REGION Network 47: ACTION IN LOADING CELL UNIT 2
   RUNG wire#powerrail
      "FC17900_MAINTENANCE_SEQUENCE"(REQUEST := 0, NUMBER_STEPS := 3, FIRST_STEP_DONE := "DB17000_MAINTENANCE_GLOBAL_VARIABLES".ACTION_DONE.POWDER.UNIT_2.HOPPER_1.LOAD_CELLS, SECOND_STEP_DONE := "DB17000_MAINTENANCE_GLOBAL_VARIABLES".ACTION_DONE.POWDER.UNIT_2.HOPPER_2.LOAD_CELLS, THRID_STEP_DONE := "DB17000_MAINTENANCE_GLOBAL_VARIABLES".ACTION_DONE.POWDER.UNIT_2.HOPPER_3.LOAD_CELLS, FOURTH_STEP_DONE := 0, FIFTH_STEP_DONE := 0, SIXTH_STEP_DONE := 0, SEVENTH_STEP_DONE := 0, FIRST_OPERATOR_HELP => "DB17100_MAINTENANCE_OPERATOR_HELP".OPERATOR_HELP[36], SECOND_OPERATOR_HELP => "DB17100_MAINTENANCE_OPERATOR_HELP".OPERATOR_HELP[41], THRID_OPERATOR_HELP => "DB17100_MAINTENANCE_OPERATOR_HELP".OPERATOR_HELP[46], FOURTH_OPERATOR_HELP => #NULL, FIFTH_OPERATOR_HELP => #NULL, SIXTH_OPERATOR_HELP => #NULL, SEVENTH_OPERATOR_HELP => #NULL, MAINTENANCE_IN_PROGRESS => "DB17200_MAINTENANCE_SEQUENCE".MAINTENANCE_IN_PROGRESS[42])
   END_RUNG
   // the same network as SCL:
   "FC17900_MAINTENANCE_SEQUENCE"(REQUEST := 0,
                           NUMBER_STEPS := 3,
                           FIRST_STEP_DONE := "DB17000_MAINTENANCE_GLOBAL_VARIABLES".ACTION_DONE.POWDER.UNIT_2.HOPPER_1.LOAD_CELLS,
                           SECOND_STEP_DONE := "DB17000_MAINTENANCE_GLOBAL_VARIABLES".ACTION_DONE.POWDER.UNIT_2.HOPPER_2.LOAD_CELLS,
                           THRID_STEP_DONE := "DB17000_MAINTENANCE_GLOBAL_VARIABLES".ACTION_DONE.POWDER.UNIT_2.HOPPER_3.LOAD_CELLS,
                           FOURTH_STEP_DONE := 0,
                           FIFTH_STEP_DONE := 0,
                           SIXTH_STEP_DONE := 0,
                           SEVENTH_STEP_DONE := 0,
                           FIRST_OPERATOR_HELP => "DB17100_MAINTENANCE_OPERATOR_HELP".OPERATOR_HELP[36],
                           SECOND_OPERATOR_HELP => "DB17100_MAINTENANCE_OPERATOR_HELP".OPERATOR_HELP[41],
                           THRID_OPERATOR_HELP => "DB17100_MAINTENANCE_OPERATOR_HELP".OPERATOR_HELP[46],
                           FOURTH_OPERATOR_HELP => #NULL,
                           FIFTH_OPERATOR_HELP => #NULL,
                           SIXTH_OPERATOR_HELP => #NULL,
                           SEVENTH_OPERATOR_HELP => #NULL,
                           MAINTENANCE_IN_PROGRESS => "DB17200_MAINTENANCE_SEQUENCE".MAINTENANCE_IN_PROGRESS[42]);
END_REGION

REGION Network 48: COMPLETE CHANGE OF FEEDER UNIT 1
   RUNG wire#powerrail
      "FC17900_MAINTENANCE_SEQUENCE"(REQUEST := 0, NUMBER_STEPS := 3, FIRST_STEP_DONE := "DB17000_MAINTENANCE_GLOBAL_VARIABLES".ACTION_DONE.POWDER.UNIT_1.FEEDER_1.TIGHTNESS_TEST_L1, SECOND_STEP_DONE := "DB17000_MAINTENANCE_GLOBAL_VARIABLES".ACTION_DONE.POWDER.UNIT_1.FEEDER_1.TIGHTNESS_TEST_L2, THRID_STEP_DONE := "DB17000_MAINTENANCE_GLOBAL_VARIABLES".ACTION_DONE.POWDER.UNIT_1.GENERAL.POWDER_FLOW_OBTAINING, FOURTH_STEP_DONE := 0, FIFTH_STEP_DONE := 0, SIXTH_STEP_DONE := 0, SEVENTH_STEP_DONE := 0, FIRST_OPERATOR_HELP => "DB17100_MAINTENANCE_OPERATOR_HELP".OPERATOR_HELP[22], SECOND_OPERATOR_HELP => "DB17100_MAINTENANCE_OPERATOR_HELP".OPERATOR_HELP[23], THRID_OPERATOR_HELP => "DB17100_MAINTENANCE_OPERATOR_HELP".OPERATOR_HELP[6], FOURTH_OPERATOR_HELP => #NULL, FIFTH_OPERATOR_HELP => #NULL, SIXTH_OPERATOR_HELP => #NULL, SEVENTH_OPERATOR_HELP => #NULL, MAINTENANCE_IN_PROGRESS => "DB17200_MAINTENANCE_SEQUENCE".MAINTENANCE_IN_PROGRESS[43])
   END_RUNG
   // the same network as SCL:
   "FC17900_MAINTENANCE_SEQUENCE"(REQUEST := 0,
                           NUMBER_STEPS := 3,
                           FIRST_STEP_DONE := "DB17000_MAINTENANCE_GLOBAL_VARIABLES".ACTION_DONE.POWDER.UNIT_1.FEEDER_1.TIGHTNESS_TEST_L1,
                           SECOND_STEP_DONE := "DB17000_MAINTENANCE_GLOBAL_VARIABLES".ACTION_DONE.POWDER.UNIT_1.FEEDER_1.TIGHTNESS_TEST_L2,
                           THRID_STEP_DONE := "DB17000_MAINTENANCE_GLOBAL_VARIABLES".ACTION_DONE.POWDER.UNIT_1.GENERAL.POWDER_FLOW_OBTAINING,
                           FOURTH_STEP_DONE := 0,
                           FIFTH_STEP_DONE := 0,
                           SIXTH_STEP_DONE := 0,
                           SEVENTH_STEP_DONE := 0,
                           FIRST_OPERATOR_HELP => "DB17100_MAINTENANCE_OPERATOR_HELP".OPERATOR_HELP[22],
                           SECOND_OPERATOR_HELP => "DB17100_MAINTENANCE_OPERATOR_HELP".OPERATOR_HELP[23],
                           THRID_OPERATOR_HELP => "DB17100_MAINTENANCE_OPERATOR_HELP".OPERATOR_HELP[6],
                           FOURTH_OPERATOR_HELP => #NULL,
                           FIFTH_OPERATOR_HELP => #NULL,
                           SIXTH_OPERATOR_HELP => #NULL,
                           SEVENTH_OPERATOR_HELP => #NULL,
                           MAINTENANCE_IN_PROGRESS => "DB17200_MAINTENANCE_SEQUENCE".MAINTENANCE_IN_PROGRESS[43]);
END_REGION

REGION Network 49: COMPLETE CHANGE OF FEEDER UNIT 2
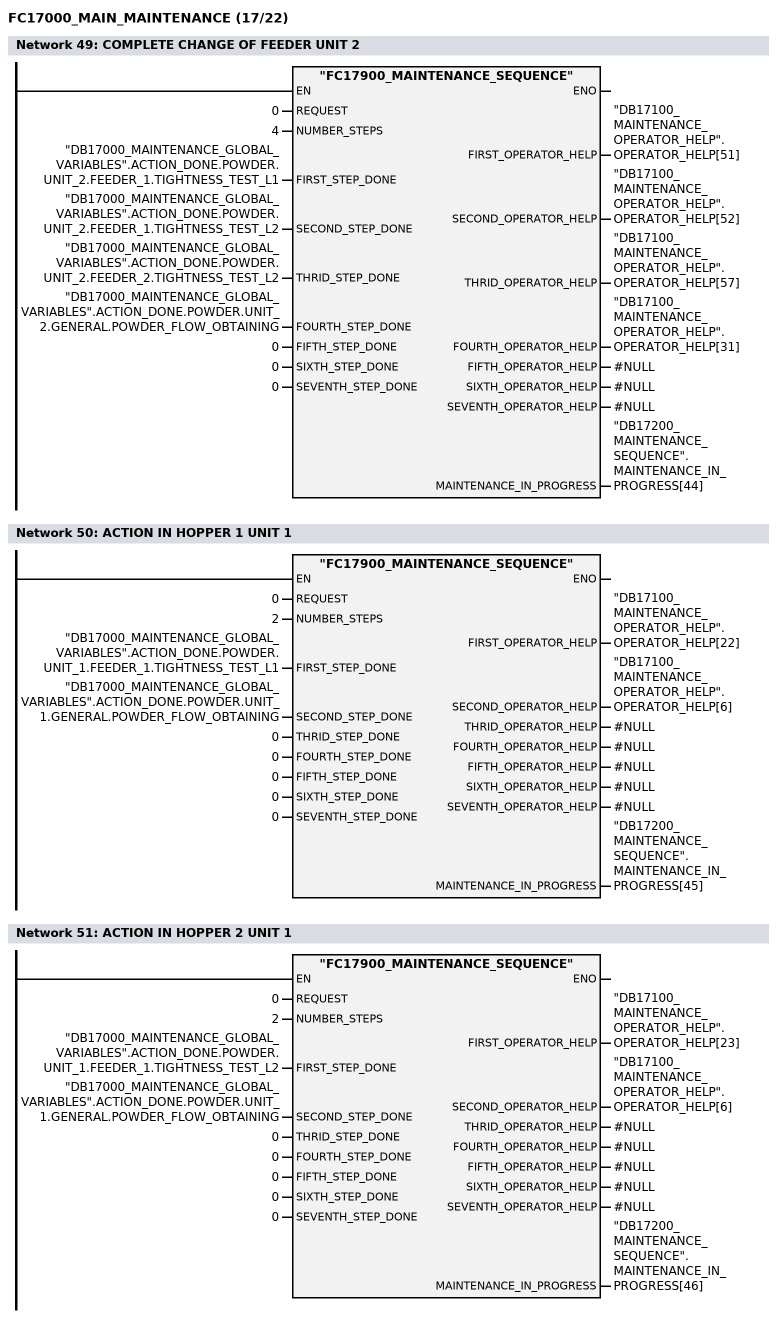
   RUNG wire#powerrail
      "FC17900_MAINTENANCE_SEQUENCE"(REQUEST := 0, NUMBER_STEPS := 4, FIRST_STEP_DONE := "DB17000_MAINTENANCE_GLOBAL_VARIABLES".ACTION_DONE.POWDER.UNIT_2.FEEDER_1.TIGHTNESS_TEST_L1, SECOND_STEP_DONE := "DB17000_MAINTENANCE_GLOBAL_VARIABLES".ACTION_DONE.POWDER.UNIT_2.FEEDER_1.TIGHTNESS_TEST_L2, THRID_STEP_DONE := "DB17000_MAINTENANCE_GLOBAL_VARIABLES".ACTION_DONE.POWDER.UNIT_2.FEEDER_2.TIGHTNESS_TEST_L2, FOURTH_STEP_DONE := "DB17000_MAINTENANCE_GLOBAL_VARIABLES".ACTION_DONE.POWDER.UNIT_2.GENERAL.POWDER_FLOW_OBTAINING, FIFTH_STEP_DONE := 0, SIXTH_STEP_DONE := 0, SEVENTH_STEP_DONE := 0, FIRST_OPERATOR_HELP => "DB17100_MAINTENANCE_OPERATOR_HELP".OPERATOR_HELP[51], SECOND_OPERATOR_HELP => "DB17100_MAINTENANCE_OPERATOR_HELP".OPERATOR_HELP[52], THRID_OPERATOR_HELP => "DB17100_MAINTENANCE_OPERATOR_HELP".OPERATOR_HELP[57], FOURTH_OPERATOR_HELP => "DB17100_MAINTENANCE_OPERATOR_HELP".OPERATOR_HELP[31], FIFTH_OPERATOR_HELP => #NULL, SIXTH_OPERATOR_HELP => #NULL, SEVENTH_OPERATOR_HELP => #NULL, MAINTENANCE_IN_PROGRESS => "DB17200_MAINTENANCE_SEQUENCE".MAINTENANCE_IN_PROGRESS[44])
   END_RUNG
   // the same network as SCL:
   "FC17900_MAINTENANCE_SEQUENCE"(REQUEST := 0,
                           NUMBER_STEPS := 4,
                           FIRST_STEP_DONE := "DB17000_MAINTENANCE_GLOBAL_VARIABLES".ACTION_DONE.POWDER.UNIT_2.FEEDER_1.TIGHTNESS_TEST_L1,
                           SECOND_STEP_DONE := "DB17000_MAINTENANCE_GLOBAL_VARIABLES".ACTION_DONE.POWDER.UNIT_2.FEEDER_1.TIGHTNESS_TEST_L2,
                           THRID_STEP_DONE := "DB17000_MAINTENANCE_GLOBAL_VARIABLES".ACTION_DONE.POWDER.UNIT_2.FEEDER_2.TIGHTNESS_TEST_L2,
                           FOURTH_STEP_DONE := "DB17000_MAINTENANCE_GLOBAL_VARIABLES".ACTION_DONE.POWDER.UNIT_2.GENERAL.POWDER_FLOW_OBTAINING,
                           FIFTH_STEP_DONE := 0,
                           SIXTH_STEP_DONE := 0,
                           SEVENTH_STEP_DONE := 0,
                           FIRST_OPERATOR_HELP => "DB17100_MAINTENANCE_OPERATOR_HELP".OPERATOR_HELP[51],
                           SECOND_OPERATOR_HELP => "DB17100_MAINTENANCE_OPERATOR_HELP".OPERATOR_HELP[52],
                           THRID_OPERATOR_HELP => "DB17100_MAINTENANCE_OPERATOR_HELP".OPERATOR_HELP[57],
                           FOURTH_OPERATOR_HELP => "DB17100_MAINTENANCE_OPERATOR_HELP".OPERATOR_HELP[31],
                           FIFTH_OPERATOR_HELP => #NULL,
                           SIXTH_OPERATOR_HELP => #NULL,
                           SEVENTH_OPERATOR_HELP => #NULL,
                           MAINTENANCE_IN_PROGRESS => "DB17200_MAINTENANCE_SEQUENCE".MAINTENANCE_IN_PROGRESS[44]);
END_REGION

REGION Network 50: ACTION IN HOPPER 1 UNIT 1
   RUNG wire#powerrail
      "FC17900_MAINTENANCE_SEQUENCE"(REQUEST := 0, NUMBER_STEPS := 2, FIRST_STEP_DONE := "DB17000_MAINTENANCE_GLOBAL_VARIABLES".ACTION_DONE.POWDER.UNIT_1.FEEDER_1.TIGHTNESS_TEST_L1, SECOND_STEP_DONE := "DB17000_MAINTENANCE_GLOBAL_VARIABLES".ACTION_DONE.POWDER.UNIT_1.GENERAL.POWDER_FLOW_OBTAINING, THRID_STEP_DONE := 0, FOURTH_STEP_DONE := 0, FIFTH_STEP_DONE := 0, SIXTH_STEP_DONE := 0, SEVENTH_STEP_DONE := 0, FIRST_OPERATOR_HELP => "DB17100_MAINTENANCE_OPERATOR_HELP".OPERATOR_HELP[22], SECOND_OPERATOR_HELP => "DB17100_MAINTENANCE_OPERATOR_HELP".OPERATOR_HELP[6], THRID_OPERATOR_HELP => #NULL, FOURTH_OPERATOR_HELP => #NULL, FIFTH_OPERATOR_HELP => #NULL, SIXTH_OPERATOR_HELP => #NULL, SEVENTH_OPERATOR_HELP => #NULL, MAINTENANCE_IN_PROGRESS => "DB17200_MAINTENANCE_SEQUENCE".MAINTENANCE_IN_PROGRESS[45])
   END_RUNG
   // the same network as SCL:
   "FC17900_MAINTENANCE_SEQUENCE"(REQUEST := 0,
                           NUMBER_STEPS := 2,
                           FIRST_STEP_DONE := "DB17000_MAINTENANCE_GLOBAL_VARIABLES".ACTION_DONE.POWDER.UNIT_1.FEEDER_1.TIGHTNESS_TEST_L1,
                           SECOND_STEP_DONE := "DB17000_MAINTENANCE_GLOBAL_VARIABLES".ACTION_DONE.POWDER.UNIT_1.GENERAL.POWDER_FLOW_OBTAINING,
                           THRID_STEP_DONE := 0,
                           FOURTH_STEP_DONE := 0,
                           FIFTH_STEP_DONE := 0,
                           SIXTH_STEP_DONE := 0,
                           SEVENTH_STEP_DONE := 0,
                           FIRST_OPERATOR_HELP => "DB17100_MAINTENANCE_OPERATOR_HELP".OPERATOR_HELP[22],
                           SECOND_OPERATOR_HELP => "DB17100_MAINTENANCE_OPERATOR_HELP".OPERATOR_HELP[6],
                           THRID_OPERATOR_HELP => #NULL,
                           FOURTH_OPERATOR_HELP => #NULL,
                           FIFTH_OPERATOR_HELP => #NULL,
                           SIXTH_OPERATOR_HELP => #NULL,
                           SEVENTH_OPERATOR_HELP => #NULL,
                           MAINTENANCE_IN_PROGRESS => "DB17200_MAINTENANCE_SEQUENCE".MAINTENANCE_IN_PROGRESS[45]);
END_REGION

REGION Network 51: ACTION IN HOPPER 2 UNIT 1
   RUNG wire#powerrail
      "FC17900_MAINTENANCE_SEQUENCE"(REQUEST := 0, NUMBER_STEPS := 2, FIRST_STEP_DONE := "DB17000_MAINTENANCE_GLOBAL_VARIABLES".ACTION_DONE.POWDER.UNIT_1.FEEDER_1.TIGHTNESS_TEST_L2, SECOND_STEP_DONE := "DB17000_MAINTENANCE_GLOBAL_VARIABLES".ACTION_DONE.POWDER.UNIT_1.GENERAL.POWDER_FLOW_OBTAINING, THRID_STEP_DONE := 0, FOURTH_STEP_DONE := 0, FIFTH_STEP_DONE := 0, SIXTH_STEP_DONE := 0, SEVENTH_STEP_DONE := 0, FIRST_OPERATOR_HELP => "DB17100_MAINTENANCE_OPERATOR_HELP".OPERATOR_HELP[23], SECOND_OPERATOR_HELP => "DB17100_MAINTENANCE_OPERATOR_HELP".OPERATOR_HELP[6], THRID_OPERATOR_HELP => #NULL, FOURTH_OPERATOR_HELP => #NULL, FIFTH_OPERATOR_HELP => #NULL, SIXTH_OPERATOR_HELP => #NULL, SEVENTH_OPERATOR_HELP => #NULL, MAINTENANCE_IN_PROGRESS => "DB17200_MAINTENANCE_SEQUENCE".MAINTENANCE_IN_PROGRESS[46])
   END_RUNG
   // the same network as SCL:
   "FC17900_MAINTENANCE_SEQUENCE"(REQUEST := 0,
                           NUMBER_STEPS := 2,
                           FIRST_STEP_DONE := "DB17000_MAINTENANCE_GLOBAL_VARIABLES".ACTION_DONE.POWDER.UNIT_1.FEEDER_1.TIGHTNESS_TEST_L2,
                           SECOND_STEP_DONE := "DB17000_MAINTENANCE_GLOBAL_VARIABLES".ACTION_DONE.POWDER.UNIT_1.GENERAL.POWDER_FLOW_OBTAINING,
                           THRID_STEP_DONE := 0,
                           FOURTH_STEP_DONE := 0,
                           FIFTH_STEP_DONE := 0,
                           SIXTH_STEP_DONE := 0,
                           SEVENTH_STEP_DONE := 0,
                           FIRST_OPERATOR_HELP => "DB17100_MAINTENANCE_OPERATOR_HELP".OPERATOR_HELP[23],
                           SECOND_OPERATOR_HELP => "DB17100_MAINTENANCE_OPERATOR_HELP".OPERATOR_HELP[6],
                           THRID_OPERATOR_HELP => #NULL,
                           FOURTH_OPERATOR_HELP => #NULL,
                           FIFTH_OPERATOR_HELP => #NULL,
                           SIXTH_OPERATOR_HELP => #NULL,
                           SEVENTH_OPERATOR_HELP => #NULL,
                           MAINTENANCE_IN_PROGRESS => "DB17200_MAINTENANCE_SEQUENCE".MAINTENANCE_IN_PROGRESS[46]);
END_REGION

REGION Network 52: ACTION IN HOPPER 1 UNIT 2
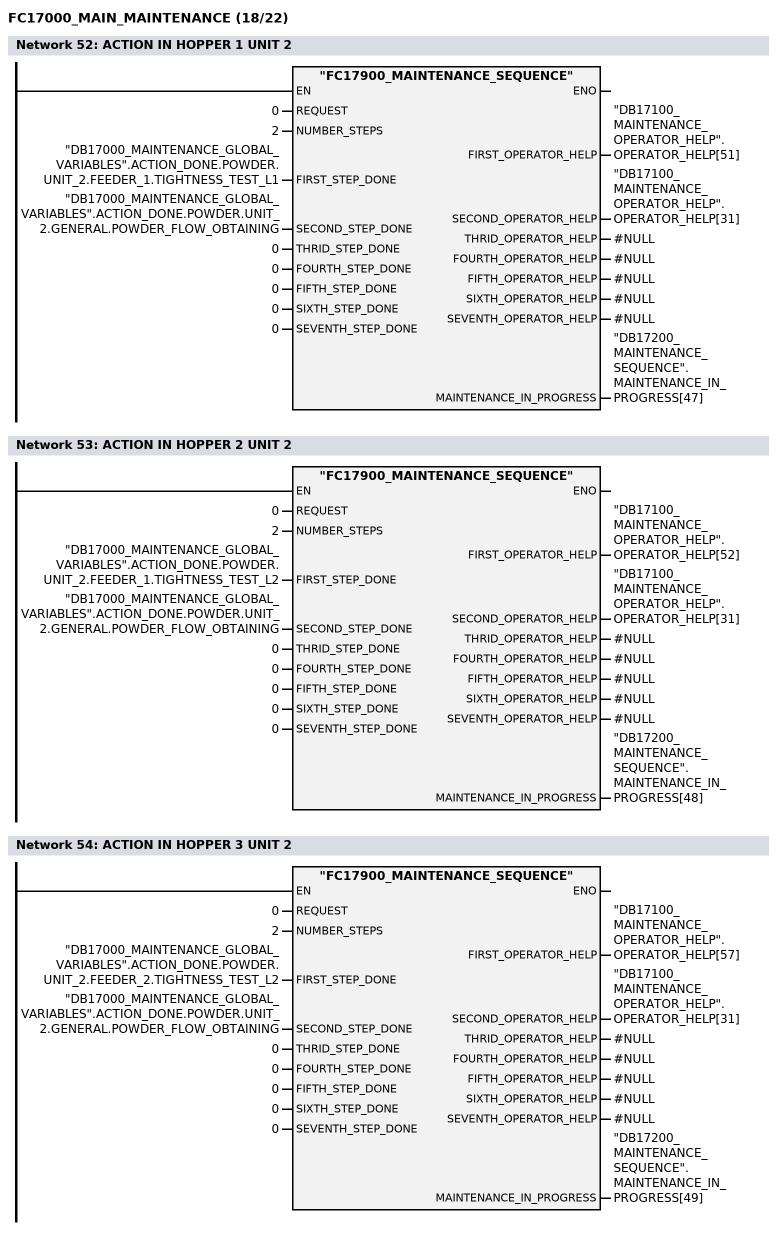
   RUNG wire#powerrail
      "FC17900_MAINTENANCE_SEQUENCE"(REQUEST := 0, NUMBER_STEPS := 2, FIRST_STEP_DONE := "DB17000_MAINTENANCE_GLOBAL_VARIABLES".ACTION_DONE.POWDER.UNIT_2.FEEDER_1.TIGHTNESS_TEST_L1, SECOND_STEP_DONE := "DB17000_MAINTENANCE_GLOBAL_VARIABLES".ACTION_DONE.POWDER.UNIT_2.GENERAL.POWDER_FLOW_OBTAINING, THRID_STEP_DONE := 0, FOURTH_STEP_DONE := 0, FIFTH_STEP_DONE := 0, SIXTH_STEP_DONE := 0, SEVENTH_STEP_DONE := 0, FIRST_OPERATOR_HELP => "DB17100_MAINTENANCE_OPERATOR_HELP".OPERATOR_HELP[51], SECOND_OPERATOR_HELP => "DB17100_MAINTENANCE_OPERATOR_HELP".OPERATOR_HELP[31], THRID_OPERATOR_HELP => #NULL, FOURTH_OPERATOR_HELP => #NULL, FIFTH_OPERATOR_HELP => #NULL, SIXTH_OPERATOR_HELP => #NULL, SEVENTH_OPERATOR_HELP => #NULL, MAINTENANCE_IN_PROGRESS => "DB17200_MAINTENANCE_SEQUENCE".MAINTENANCE_IN_PROGRESS[47])
   END_RUNG
   // the same network as SCL:
   "FC17900_MAINTENANCE_SEQUENCE"(REQUEST := 0,
                           NUMBER_STEPS := 2,
                           FIRST_STEP_DONE := "DB17000_MAINTENANCE_GLOBAL_VARIABLES".ACTION_DONE.POWDER.UNIT_2.FEEDER_1.TIGHTNESS_TEST_L1,
                           SECOND_STEP_DONE := "DB17000_MAINTENANCE_GLOBAL_VARIABLES".ACTION_DONE.POWDER.UNIT_2.GENERAL.POWDER_FLOW_OBTAINING,
                           THRID_STEP_DONE := 0,
                           FOURTH_STEP_DONE := 0,
                           FIFTH_STEP_DONE := 0,
                           SIXTH_STEP_DONE := 0,
                           SEVENTH_STEP_DONE := 0,
                           FIRST_OPERATOR_HELP => "DB17100_MAINTENANCE_OPERATOR_HELP".OPERATOR_HELP[51],
                           SECOND_OPERATOR_HELP => "DB17100_MAINTENANCE_OPERATOR_HELP".OPERATOR_HELP[31],
                           THRID_OPERATOR_HELP => #NULL,
                           FOURTH_OPERATOR_HELP => #NULL,
                           FIFTH_OPERATOR_HELP => #NULL,
                           SIXTH_OPERATOR_HELP => #NULL,
                           SEVENTH_OPERATOR_HELP => #NULL,
                           MAINTENANCE_IN_PROGRESS => "DB17200_MAINTENANCE_SEQUENCE".MAINTENANCE_IN_PROGRESS[47]);
END_REGION

REGION Network 53: ACTION IN HOPPER 2 UNIT 2
   RUNG wire#powerrail
      "FC17900_MAINTENANCE_SEQUENCE"(REQUEST := 0, NUMBER_STEPS := 2, FIRST_STEP_DONE := "DB17000_MAINTENANCE_GLOBAL_VARIABLES".ACTION_DONE.POWDER.UNIT_2.FEEDER_1.TIGHTNESS_TEST_L2, SECOND_STEP_DONE := "DB17000_MAINTENANCE_GLOBAL_VARIABLES".ACTION_DONE.POWDER.UNIT_2.GENERAL.POWDER_FLOW_OBTAINING, THRID_STEP_DONE := 0, FOURTH_STEP_DONE := 0, FIFTH_STEP_DONE := 0, SIXTH_STEP_DONE := 0, SEVENTH_STEP_DONE := 0, FIRST_OPERATOR_HELP => "DB17100_MAINTENANCE_OPERATOR_HELP".OPERATOR_HELP[52], SECOND_OPERATOR_HELP => "DB17100_MAINTENANCE_OPERATOR_HELP".OPERATOR_HELP[31], THRID_OPERATOR_HELP => #NULL, FOURTH_OPERATOR_HELP => #NULL, FIFTH_OPERATOR_HELP => #NULL, SIXTH_OPERATOR_HELP => #NULL, SEVENTH_OPERATOR_HELP => #NULL, MAINTENANCE_IN_PROGRESS => "DB17200_MAINTENANCE_SEQUENCE".MAINTENANCE_IN_PROGRESS[48])
   END_RUNG
   // the same network as SCL:
   "FC17900_MAINTENANCE_SEQUENCE"(REQUEST := 0,
                           NUMBER_STEPS := 2,
                           FIRST_STEP_DONE := "DB17000_MAINTENANCE_GLOBAL_VARIABLES".ACTION_DONE.POWDER.UNIT_2.FEEDER_1.TIGHTNESS_TEST_L2,
                           SECOND_STEP_DONE := "DB17000_MAINTENANCE_GLOBAL_VARIABLES".ACTION_DONE.POWDER.UNIT_2.GENERAL.POWDER_FLOW_OBTAINING,
                           THRID_STEP_DONE := 0,
                           FOURTH_STEP_DONE := 0,
                           FIFTH_STEP_DONE := 0,
                           SIXTH_STEP_DONE := 0,
                           SEVENTH_STEP_DONE := 0,
                           FIRST_OPERATOR_HELP => "DB17100_MAINTENANCE_OPERATOR_HELP".OPERATOR_HELP[52],
                           SECOND_OPERATOR_HELP => "DB17100_MAINTENANCE_OPERATOR_HELP".OPERATOR_HELP[31],
                           THRID_OPERATOR_HELP => #NULL,
                           FOURTH_OPERATOR_HELP => #NULL,
                           FIFTH_OPERATOR_HELP => #NULL,
                           SIXTH_OPERATOR_HELP => #NULL,
                           SEVENTH_OPERATOR_HELP => #NULL,
                           MAINTENANCE_IN_PROGRESS => "DB17200_MAINTENANCE_SEQUENCE".MAINTENANCE_IN_PROGRESS[48]);
END_REGION

REGION Network 54: ACTION IN HOPPER 3 UNIT 2
   RUNG wire#powerrail
      "FC17900_MAINTENANCE_SEQUENCE"(REQUEST := 0, NUMBER_STEPS := 2, FIRST_STEP_DONE := "DB17000_MAINTENANCE_GLOBAL_VARIABLES".ACTION_DONE.POWDER.UNIT_2.FEEDER_2.TIGHTNESS_TEST_L2, SECOND_STEP_DONE := "DB17000_MAINTENANCE_GLOBAL_VARIABLES".ACTION_DONE.POWDER.UNIT_2.GENERAL.POWDER_FLOW_OBTAINING, THRID_STEP_DONE := 0, FOURTH_STEP_DONE := 0, FIFTH_STEP_DONE := 0, SIXTH_STEP_DONE := 0, SEVENTH_STEP_DONE := 0, FIRST_OPERATOR_HELP => "DB17100_MAINTENANCE_OPERATOR_HELP".OPERATOR_HELP[57], SECOND_OPERATOR_HELP => "DB17100_MAINTENANCE_OPERATOR_HELP".OPERATOR_HELP[31], THRID_OPERATOR_HELP => #NULL, FOURTH_OPERATOR_HELP => #NULL, FIFTH_OPERATOR_HELP => #NULL, SIXTH_OPERATOR_HELP => #NULL, SEVENTH_OPERATOR_HELP => #NULL, MAINTENANCE_IN_PROGRESS => "DB17200_MAINTENANCE_SEQUENCE".MAINTENANCE_IN_PROGRESS[49])
   END_RUNG
   // the same network as SCL:
   "FC17900_MAINTENANCE_SEQUENCE"(REQUEST := 0,
                           NUMBER_STEPS := 2,
                           FIRST_STEP_DONE := "DB17000_MAINTENANCE_GLOBAL_VARIABLES".ACTION_DONE.POWDER.UNIT_2.FEEDER_2.TIGHTNESS_TEST_L2,
                           SECOND_STEP_DONE := "DB17000_MAINTENANCE_GLOBAL_VARIABLES".ACTION_DONE.POWDER.UNIT_2.GENERAL.POWDER_FLOW_OBTAINING,
                           THRID_STEP_DONE := 0,
                           FOURTH_STEP_DONE := 0,
                           FIFTH_STEP_DONE := 0,
                           SIXTH_STEP_DONE := 0,
                           SEVENTH_STEP_DONE := 0,
                           FIRST_OPERATOR_HELP => "DB17100_MAINTENANCE_OPERATOR_HELP".OPERATOR_HELP[57],
                           SECOND_OPERATOR_HELP => "DB17100_MAINTENANCE_OPERATOR_HELP".OPERATOR_HELP[31],
                           THRID_OPERATOR_HELP => #NULL,
                           FOURTH_OPERATOR_HELP => #NULL,
                           FIFTH_OPERATOR_HELP => #NULL,
                           SIXTH_OPERATOR_HELP => #NULL,
                           SEVENTH_OPERATOR_HELP => #NULL,
                           MAINTENANCE_IN_PROGRESS => "DB17200_MAINTENANCE_SEQUENCE".MAINTENANCE_IN_PROGRESS[49]);
END_REGION

REGION Network 55: ACTION IN TUBE SECTION 3 LINE 1 UNIT 1
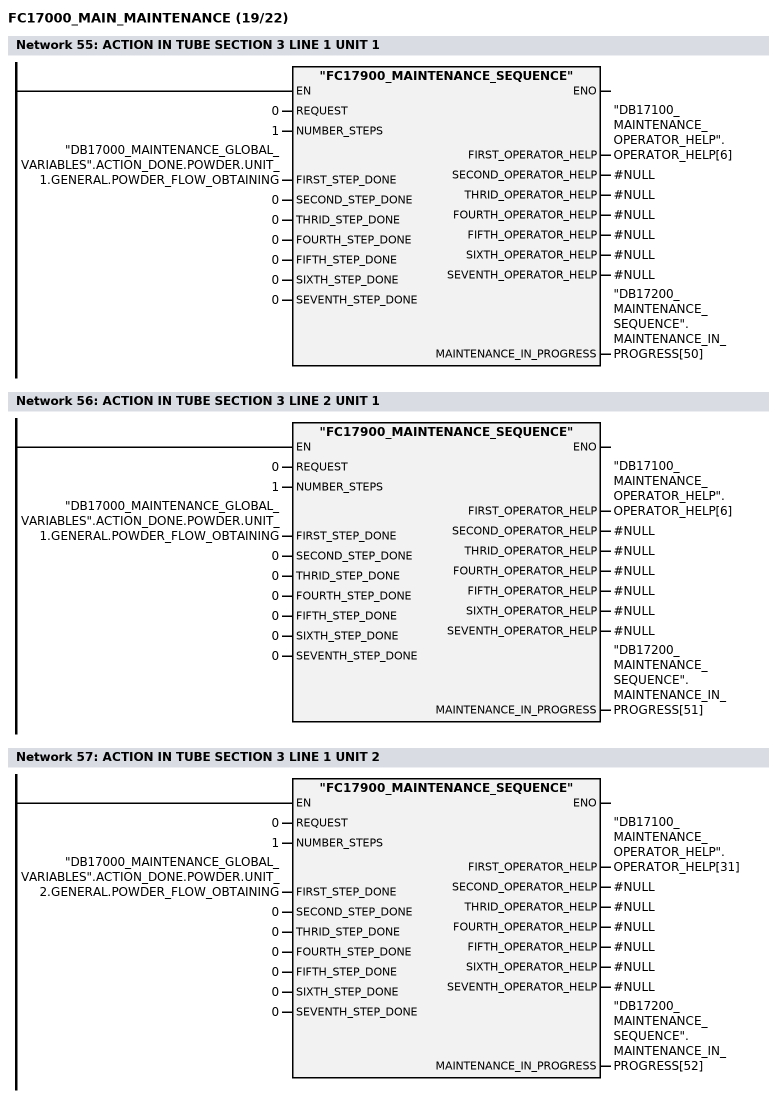
   RUNG wire#powerrail
      "FC17900_MAINTENANCE_SEQUENCE"(REQUEST := 0, NUMBER_STEPS := 1, FIRST_STEP_DONE := "DB17000_MAINTENANCE_GLOBAL_VARIABLES".ACTION_DONE.POWDER.UNIT_1.GENERAL.POWDER_FLOW_OBTAINING, SECOND_STEP_DONE := 0, THRID_STEP_DONE := 0, FOURTH_STEP_DONE := 0, FIFTH_STEP_DONE := 0, SIXTH_STEP_DONE := 0, SEVENTH_STEP_DONE := 0, FIRST_OPERATOR_HELP => "DB17100_MAINTENANCE_OPERATOR_HELP".OPERATOR_HELP[6], SECOND_OPERATOR_HELP => #NULL, THRID_OPERATOR_HELP => #NULL, FOURTH_OPERATOR_HELP => #NULL, FIFTH_OPERATOR_HELP => #NULL, SIXTH_OPERATOR_HELP => #NULL, SEVENTH_OPERATOR_HELP => #NULL, MAINTENANCE_IN_PROGRESS => "DB17200_MAINTENANCE_SEQUENCE".MAINTENANCE_IN_PROGRESS[50])
   END_RUNG
   // the same network as SCL:
   "FC17900_MAINTENANCE_SEQUENCE"(REQUEST := 0,
                           NUMBER_STEPS := 1,
                           FIRST_STEP_DONE := "DB17000_MAINTENANCE_GLOBAL_VARIABLES".ACTION_DONE.POWDER.UNIT_1.GENERAL.POWDER_FLOW_OBTAINING,
                           SECOND_STEP_DONE := 0,
                           THRID_STEP_DONE := 0,
                           FOURTH_STEP_DONE := 0,
                           FIFTH_STEP_DONE := 0,
                           SIXTH_STEP_DONE := 0,
                           SEVENTH_STEP_DONE := 0,
                           FIRST_OPERATOR_HELP => "DB17100_MAINTENANCE_OPERATOR_HELP".OPERATOR_HELP[6],
                           SECOND_OPERATOR_HELP => #NULL,
                           THRID_OPERATOR_HELP => #NULL,
                           FOURTH_OPERATOR_HELP => #NULL,
                           FIFTH_OPERATOR_HELP => #NULL,
                           SIXTH_OPERATOR_HELP => #NULL,
                           SEVENTH_OPERATOR_HELP => #NULL,
                           MAINTENANCE_IN_PROGRESS => "DB17200_MAINTENANCE_SEQUENCE".MAINTENANCE_IN_PROGRESS[50]);
END_REGION

REGION Network 56: ACTION IN TUBE SECTION 3 LINE 2 UNIT 1
   RUNG wire#powerrail
      "FC17900_MAINTENANCE_SEQUENCE"(REQUEST := 0, NUMBER_STEPS := 1, FIRST_STEP_DONE := "DB17000_MAINTENANCE_GLOBAL_VARIABLES".ACTION_DONE.POWDER.UNIT_1.GENERAL.POWDER_FLOW_OBTAINING, SECOND_STEP_DONE := 0, THRID_STEP_DONE := 0, FOURTH_STEP_DONE := 0, FIFTH_STEP_DONE := 0, SIXTH_STEP_DONE := 0, SEVENTH_STEP_DONE := 0, FIRST_OPERATOR_HELP => "DB17100_MAINTENANCE_OPERATOR_HELP".OPERATOR_HELP[6], SECOND_OPERATOR_HELP => #NULL, THRID_OPERATOR_HELP => #NULL, FOURTH_OPERATOR_HELP => #NULL, FIFTH_OPERATOR_HELP => #NULL, SIXTH_OPERATOR_HELP => #NULL, SEVENTH_OPERATOR_HELP => #NULL, MAINTENANCE_IN_PROGRESS => "DB17200_MAINTENANCE_SEQUENCE".MAINTENANCE_IN_PROGRESS[51])
   END_RUNG
   // the same network as SCL:
   "FC17900_MAINTENANCE_SEQUENCE"(REQUEST := 0,
                           NUMBER_STEPS := 1,
                           FIRST_STEP_DONE := "DB17000_MAINTENANCE_GLOBAL_VARIABLES".ACTION_DONE.POWDER.UNIT_1.GENERAL.POWDER_FLOW_OBTAINING,
                           SECOND_STEP_DONE := 0,
                           THRID_STEP_DONE := 0,
                           FOURTH_STEP_DONE := 0,
                           FIFTH_STEP_DONE := 0,
                           SIXTH_STEP_DONE := 0,
                           SEVENTH_STEP_DONE := 0,
                           FIRST_OPERATOR_HELP => "DB17100_MAINTENANCE_OPERATOR_HELP".OPERATOR_HELP[6],
                           SECOND_OPERATOR_HELP => #NULL,
                           THRID_OPERATOR_HELP => #NULL,
                           FOURTH_OPERATOR_HELP => #NULL,
                           FIFTH_OPERATOR_HELP => #NULL,
                           SIXTH_OPERATOR_HELP => #NULL,
                           SEVENTH_OPERATOR_HELP => #NULL,
                           MAINTENANCE_IN_PROGRESS => "DB17200_MAINTENANCE_SEQUENCE".MAINTENANCE_IN_PROGRESS[51]);
END_REGION

REGION Network 57: ACTION IN TUBE SECTION 3 LINE 1 UNIT 2
   RUNG wire#powerrail
      "FC17900_MAINTENANCE_SEQUENCE"(REQUEST := 0, NUMBER_STEPS := 1, FIRST_STEP_DONE := "DB17000_MAINTENANCE_GLOBAL_VARIABLES".ACTION_DONE.POWDER.UNIT_2.GENERAL.POWDER_FLOW_OBTAINING, SECOND_STEP_DONE := 0, THRID_STEP_DONE := 0, FOURTH_STEP_DONE := 0, FIFTH_STEP_DONE := 0, SIXTH_STEP_DONE := 0, SEVENTH_STEP_DONE := 0, FIRST_OPERATOR_HELP => "DB17100_MAINTENANCE_OPERATOR_HELP".OPERATOR_HELP[31], SECOND_OPERATOR_HELP => #NULL, THRID_OPERATOR_HELP => #NULL, FOURTH_OPERATOR_HELP => #NULL, FIFTH_OPERATOR_HELP => #NULL, SIXTH_OPERATOR_HELP => #NULL, SEVENTH_OPERATOR_HELP => #NULL, MAINTENANCE_IN_PROGRESS => "DB17200_MAINTENANCE_SEQUENCE".MAINTENANCE_IN_PROGRESS[52])
   END_RUNG
   // the same network as SCL:
   "FC17900_MAINTENANCE_SEQUENCE"(REQUEST := 0,
                           NUMBER_STEPS := 1,
                           FIRST_STEP_DONE := "DB17000_MAINTENANCE_GLOBAL_VARIABLES".ACTION_DONE.POWDER.UNIT_2.GENERAL.POWDER_FLOW_OBTAINING,
                           SECOND_STEP_DONE := 0,
                           THRID_STEP_DONE := 0,
                           FOURTH_STEP_DONE := 0,
                           FIFTH_STEP_DONE := 0,
                           SIXTH_STEP_DONE := 0,
                           SEVENTH_STEP_DONE := 0,
                           FIRST_OPERATOR_HELP => "DB17100_MAINTENANCE_OPERATOR_HELP".OPERATOR_HELP[31],
                           SECOND_OPERATOR_HELP => #NULL,
                           THRID_OPERATOR_HELP => #NULL,
                           FOURTH_OPERATOR_HELP => #NULL,
                           FIFTH_OPERATOR_HELP => #NULL,
                           SIXTH_OPERATOR_HELP => #NULL,
                           SEVENTH_OPERATOR_HELP => #NULL,
                           MAINTENANCE_IN_PROGRESS => "DB17200_MAINTENANCE_SEQUENCE".MAINTENANCE_IN_PROGRESS[52]);
END_REGION

REGION Network 58: ACTION IN TUBE SECTION 3 LINE 2 UNIT 2
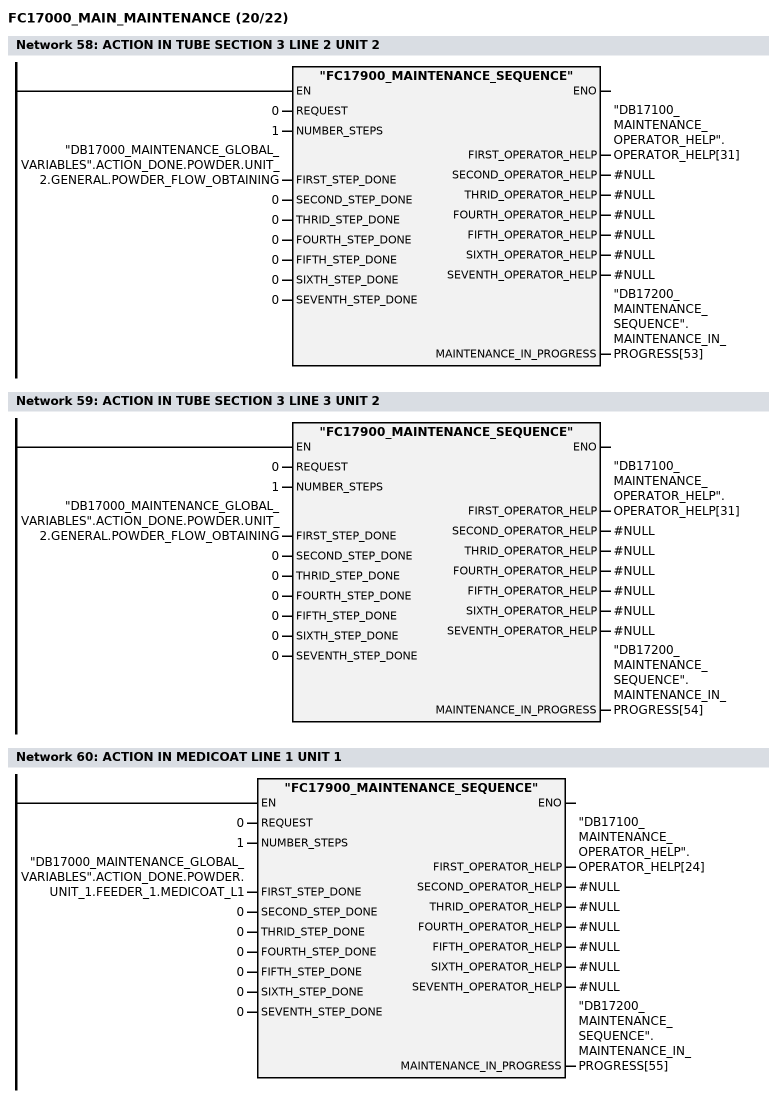
   RUNG wire#powerrail
      "FC17900_MAINTENANCE_SEQUENCE"(REQUEST := 0, NUMBER_STEPS := 1, FIRST_STEP_DONE := "DB17000_MAINTENANCE_GLOBAL_VARIABLES".ACTION_DONE.POWDER.UNIT_2.GENERAL.POWDER_FLOW_OBTAINING, SECOND_STEP_DONE := 0, THRID_STEP_DONE := 0, FOURTH_STEP_DONE := 0, FIFTH_STEP_DONE := 0, SIXTH_STEP_DONE := 0, SEVENTH_STEP_DONE := 0, FIRST_OPERATOR_HELP => "DB17100_MAINTENANCE_OPERATOR_HELP".OPERATOR_HELP[31], SECOND_OPERATOR_HELP => #NULL, THRID_OPERATOR_HELP => #NULL, FOURTH_OPERATOR_HELP => #NULL, FIFTH_OPERATOR_HELP => #NULL, SIXTH_OPERATOR_HELP => #NULL, SEVENTH_OPERATOR_HELP => #NULL, MAINTENANCE_IN_PROGRESS => "DB17200_MAINTENANCE_SEQUENCE".MAINTENANCE_IN_PROGRESS[53])
   END_RUNG
   // the same network as SCL:
   "FC17900_MAINTENANCE_SEQUENCE"(REQUEST := 0,
                           NUMBER_STEPS := 1,
                           FIRST_STEP_DONE := "DB17000_MAINTENANCE_GLOBAL_VARIABLES".ACTION_DONE.POWDER.UNIT_2.GENERAL.POWDER_FLOW_OBTAINING,
                           SECOND_STEP_DONE := 0,
                           THRID_STEP_DONE := 0,
                           FOURTH_STEP_DONE := 0,
                           FIFTH_STEP_DONE := 0,
                           SIXTH_STEP_DONE := 0,
                           SEVENTH_STEP_DONE := 0,
                           FIRST_OPERATOR_HELP => "DB17100_MAINTENANCE_OPERATOR_HELP".OPERATOR_HELP[31],
                           SECOND_OPERATOR_HELP => #NULL,
                           THRID_OPERATOR_HELP => #NULL,
                           FOURTH_OPERATOR_HELP => #NULL,
                           FIFTH_OPERATOR_HELP => #NULL,
                           SIXTH_OPERATOR_HELP => #NULL,
                           SEVENTH_OPERATOR_HELP => #NULL,
                           MAINTENANCE_IN_PROGRESS => "DB17200_MAINTENANCE_SEQUENCE".MAINTENANCE_IN_PROGRESS[53]);
END_REGION

REGION Network 59: ACTION IN TUBE SECTION 3 LINE 3 UNIT 2
   RUNG wire#powerrail
      "FC17900_MAINTENANCE_SEQUENCE"(REQUEST := 0, NUMBER_STEPS := 1, FIRST_STEP_DONE := "DB17000_MAINTENANCE_GLOBAL_VARIABLES".ACTION_DONE.POWDER.UNIT_2.GENERAL.POWDER_FLOW_OBTAINING, SECOND_STEP_DONE := 0, THRID_STEP_DONE := 0, FOURTH_STEP_DONE := 0, FIFTH_STEP_DONE := 0, SIXTH_STEP_DONE := 0, SEVENTH_STEP_DONE := 0, FIRST_OPERATOR_HELP => "DB17100_MAINTENANCE_OPERATOR_HELP".OPERATOR_HELP[31], SECOND_OPERATOR_HELP => #NULL, THRID_OPERATOR_HELP => #NULL, FOURTH_OPERATOR_HELP => #NULL, FIFTH_OPERATOR_HELP => #NULL, SIXTH_OPERATOR_HELP => #NULL, SEVENTH_OPERATOR_HELP => #NULL, MAINTENANCE_IN_PROGRESS => "DB17200_MAINTENANCE_SEQUENCE".MAINTENANCE_IN_PROGRESS[54])
   END_RUNG
   // the same network as SCL:
   "FC17900_MAINTENANCE_SEQUENCE"(REQUEST := 0,
                           NUMBER_STEPS := 1,
                           FIRST_STEP_DONE := "DB17000_MAINTENANCE_GLOBAL_VARIABLES".ACTION_DONE.POWDER.UNIT_2.GENERAL.POWDER_FLOW_OBTAINING,
                           SECOND_STEP_DONE := 0,
                           THRID_STEP_DONE := 0,
                           FOURTH_STEP_DONE := 0,
                           FIFTH_STEP_DONE := 0,
                           SIXTH_STEP_DONE := 0,
                           SEVENTH_STEP_DONE := 0,
                           FIRST_OPERATOR_HELP => "DB17100_MAINTENANCE_OPERATOR_HELP".OPERATOR_HELP[31],
                           SECOND_OPERATOR_HELP => #NULL,
                           THRID_OPERATOR_HELP => #NULL,
                           FOURTH_OPERATOR_HELP => #NULL,
                           FIFTH_OPERATOR_HELP => #NULL,
                           SIXTH_OPERATOR_HELP => #NULL,
                           SEVENTH_OPERATOR_HELP => #NULL,
                           MAINTENANCE_IN_PROGRESS => "DB17200_MAINTENANCE_SEQUENCE".MAINTENANCE_IN_PROGRESS[54]);
END_REGION

REGION Network 60: ACTION IN MEDICOAT LINE 1 UNIT 1
   RUNG wire#powerrail
      "FC17900_MAINTENANCE_SEQUENCE"(REQUEST := 0, NUMBER_STEPS := 1, FIRST_STEP_DONE := "DB17000_MAINTENANCE_GLOBAL_VARIABLES".ACTION_DONE.POWDER.UNIT_1.FEEDER_1.MEDICOAT_L1, SECOND_STEP_DONE := 0, THRID_STEP_DONE := 0, FOURTH_STEP_DONE := 0, FIFTH_STEP_DONE := 0, SIXTH_STEP_DONE := 0, SEVENTH_STEP_DONE := 0, FIRST_OPERATOR_HELP => "DB17100_MAINTENANCE_OPERATOR_HELP".OPERATOR_HELP[24], SECOND_OPERATOR_HELP => #NULL, THRID_OPERATOR_HELP => #NULL, FOURTH_OPERATOR_HELP => #NULL, FIFTH_OPERATOR_HELP => #NULL, SIXTH_OPERATOR_HELP => #NULL, SEVENTH_OPERATOR_HELP => #NULL, MAINTENANCE_IN_PROGRESS => "DB17200_MAINTENANCE_SEQUENCE".MAINTENANCE_IN_PROGRESS[55])
   END_RUNG
   // the same network as SCL:
   "FC17900_MAINTENANCE_SEQUENCE"(REQUEST := 0,
                           NUMBER_STEPS := 1,
                           FIRST_STEP_DONE := "DB17000_MAINTENANCE_GLOBAL_VARIABLES".ACTION_DONE.POWDER.UNIT_1.FEEDER_1.MEDICOAT_L1,
                           SECOND_STEP_DONE := 0,
                           THRID_STEP_DONE := 0,
                           FOURTH_STEP_DONE := 0,
                           FIFTH_STEP_DONE := 0,
                           SIXTH_STEP_DONE := 0,
                           SEVENTH_STEP_DONE := 0,
                           FIRST_OPERATOR_HELP => "DB17100_MAINTENANCE_OPERATOR_HELP".OPERATOR_HELP[24],
                           SECOND_OPERATOR_HELP => #NULL,
                           THRID_OPERATOR_HELP => #NULL,
                           FOURTH_OPERATOR_HELP => #NULL,
                           FIFTH_OPERATOR_HELP => #NULL,
                           SIXTH_OPERATOR_HELP => #NULL,
                           SEVENTH_OPERATOR_HELP => #NULL,
                           MAINTENANCE_IN_PROGRESS => "DB17200_MAINTENANCE_SEQUENCE".MAINTENANCE_IN_PROGRESS[55]);
END_REGION

REGION Network 61: ACTION IN MEDICOAT LINE 2 UNIT 1
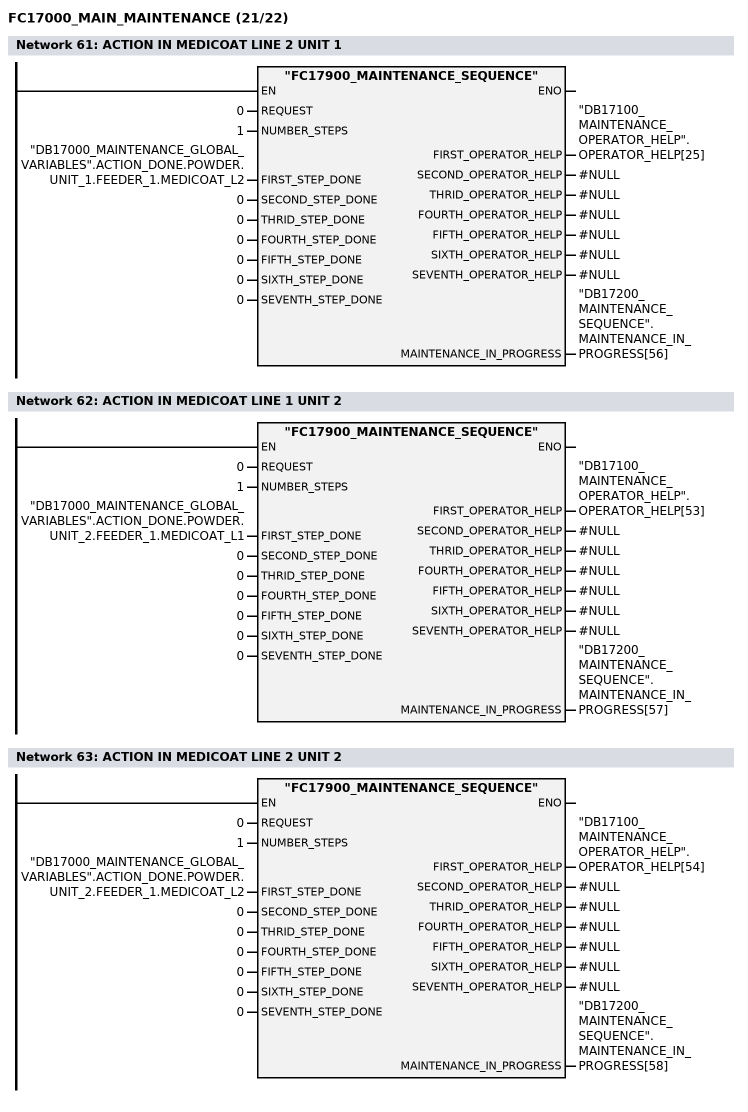
   RUNG wire#powerrail
      "FC17900_MAINTENANCE_SEQUENCE"(REQUEST := 0, NUMBER_STEPS := 1, FIRST_STEP_DONE := "DB17000_MAINTENANCE_GLOBAL_VARIABLES".ACTION_DONE.POWDER.UNIT_1.FEEDER_1.MEDICOAT_L2, SECOND_STEP_DONE := 0, THRID_STEP_DONE := 0, FOURTH_STEP_DONE := 0, FIFTH_STEP_DONE := 0, SIXTH_STEP_DONE := 0, SEVENTH_STEP_DONE := 0, FIRST_OPERATOR_HELP => "DB17100_MAINTENANCE_OPERATOR_HELP".OPERATOR_HELP[25], SECOND_OPERATOR_HELP => #NULL, THRID_OPERATOR_HELP => #NULL, FOURTH_OPERATOR_HELP => #NULL, FIFTH_OPERATOR_HELP => #NULL, SIXTH_OPERATOR_HELP => #NULL, SEVENTH_OPERATOR_HELP => #NULL, MAINTENANCE_IN_PROGRESS => "DB17200_MAINTENANCE_SEQUENCE".MAINTENANCE_IN_PROGRESS[56])
   END_RUNG
   // the same network as SCL:
   "FC17900_MAINTENANCE_SEQUENCE"(REQUEST := 0,
                           NUMBER_STEPS := 1,
                           FIRST_STEP_DONE := "DB17000_MAINTENANCE_GLOBAL_VARIABLES".ACTION_DONE.POWDER.UNIT_1.FEEDER_1.MEDICOAT_L2,
                           SECOND_STEP_DONE := 0,
                           THRID_STEP_DONE := 0,
                           FOURTH_STEP_DONE := 0,
                           FIFTH_STEP_DONE := 0,
                           SIXTH_STEP_DONE := 0,
                           SEVENTH_STEP_DONE := 0,
                           FIRST_OPERATOR_HELP => "DB17100_MAINTENANCE_OPERATOR_HELP".OPERATOR_HELP[25],
                           SECOND_OPERATOR_HELP => #NULL,
                           THRID_OPERATOR_HELP => #NULL,
                           FOURTH_OPERATOR_HELP => #NULL,
                           FIFTH_OPERATOR_HELP => #NULL,
                           SIXTH_OPERATOR_HELP => #NULL,
                           SEVENTH_OPERATOR_HELP => #NULL,
                           MAINTENANCE_IN_PROGRESS => "DB17200_MAINTENANCE_SEQUENCE".MAINTENANCE_IN_PROGRESS[56]);
END_REGION

REGION Network 62: ACTION IN MEDICOAT LINE 1 UNIT 2
   RUNG wire#powerrail
      "FC17900_MAINTENANCE_SEQUENCE"(REQUEST := 0, NUMBER_STEPS := 1, FIRST_STEP_DONE := "DB17000_MAINTENANCE_GLOBAL_VARIABLES".ACTION_DONE.POWDER.UNIT_2.FEEDER_1.MEDICOAT_L1, SECOND_STEP_DONE := 0, THRID_STEP_DONE := 0, FOURTH_STEP_DONE := 0, FIFTH_STEP_DONE := 0, SIXTH_STEP_DONE := 0, SEVENTH_STEP_DONE := 0, FIRST_OPERATOR_HELP => "DB17100_MAINTENANCE_OPERATOR_HELP".OPERATOR_HELP[53], SECOND_OPERATOR_HELP => #NULL, THRID_OPERATOR_HELP => #NULL, FOURTH_OPERATOR_HELP => #NULL, FIFTH_OPERATOR_HELP => #NULL, SIXTH_OPERATOR_HELP => #NULL, SEVENTH_OPERATOR_HELP => #NULL, MAINTENANCE_IN_PROGRESS => "DB17200_MAINTENANCE_SEQUENCE".MAINTENANCE_IN_PROGRESS[57])
   END_RUNG
   // the same network as SCL:
   "FC17900_MAINTENANCE_SEQUENCE"(REQUEST := 0,
                           NUMBER_STEPS := 1,
                           FIRST_STEP_DONE := "DB17000_MAINTENANCE_GLOBAL_VARIABLES".ACTION_DONE.POWDER.UNIT_2.FEEDER_1.MEDICOAT_L1,
                           SECOND_STEP_DONE := 0,
                           THRID_STEP_DONE := 0,
                           FOURTH_STEP_DONE := 0,
                           FIFTH_STEP_DONE := 0,
                           SIXTH_STEP_DONE := 0,
                           SEVENTH_STEP_DONE := 0,
                           FIRST_OPERATOR_HELP => "DB17100_MAINTENANCE_OPERATOR_HELP".OPERATOR_HELP[53],
                           SECOND_OPERATOR_HELP => #NULL,
                           THRID_OPERATOR_HELP => #NULL,
                           FOURTH_OPERATOR_HELP => #NULL,
                           FIFTH_OPERATOR_HELP => #NULL,
                           SIXTH_OPERATOR_HELP => #NULL,
                           SEVENTH_OPERATOR_HELP => #NULL,
                           MAINTENANCE_IN_PROGRESS => "DB17200_MAINTENANCE_SEQUENCE".MAINTENANCE_IN_PROGRESS[57]);
END_REGION

REGION Network 63: ACTION IN MEDICOAT LINE 2 UNIT 2
   RUNG wire#powerrail
      "FC17900_MAINTENANCE_SEQUENCE"(REQUEST := 0, NUMBER_STEPS := 1, FIRST_STEP_DONE := "DB17000_MAINTENANCE_GLOBAL_VARIABLES".ACTION_DONE.POWDER.UNIT_2.FEEDER_1.MEDICOAT_L2, SECOND_STEP_DONE := 0, THRID_STEP_DONE := 0, FOURTH_STEP_DONE := 0, FIFTH_STEP_DONE := 0, SIXTH_STEP_DONE := 0, SEVENTH_STEP_DONE := 0, FIRST_OPERATOR_HELP => "DB17100_MAINTENANCE_OPERATOR_HELP".OPERATOR_HELP[54], SECOND_OPERATOR_HELP => #NULL, THRID_OPERATOR_HELP => #NULL, FOURTH_OPERATOR_HELP => #NULL, FIFTH_OPERATOR_HELP => #NULL, SIXTH_OPERATOR_HELP => #NULL, SEVENTH_OPERATOR_HELP => #NULL, MAINTENANCE_IN_PROGRESS => "DB17200_MAINTENANCE_SEQUENCE".MAINTENANCE_IN_PROGRESS[58])
   END_RUNG
   // the same network as SCL:
   "FC17900_MAINTENANCE_SEQUENCE"(REQUEST := 0,
                           NUMBER_STEPS := 1,
                           FIRST_STEP_DONE := "DB17000_MAINTENANCE_GLOBAL_VARIABLES".ACTION_DONE.POWDER.UNIT_2.FEEDER_1.MEDICOAT_L2,
                           SECOND_STEP_DONE := 0,
                           THRID_STEP_DONE := 0,
                           FOURTH_STEP_DONE := 0,
                           FIFTH_STEP_DONE := 0,
                           SIXTH_STEP_DONE := 0,
                           SEVENTH_STEP_DONE := 0,
                           FIRST_OPERATOR_HELP => "DB17100_MAINTENANCE_OPERATOR_HELP".OPERATOR_HELP[54],
                           SECOND_OPERATOR_HELP => #NULL,
                           THRID_OPERATOR_HELP => #NULL,
                           FOURTH_OPERATOR_HELP => #NULL,
                           FIFTH_OPERATOR_HELP => #NULL,
                           SIXTH_OPERATOR_HELP => #NULL,
                           SEVENTH_OPERATOR_HELP => #NULL,
                           MAINTENANCE_IN_PROGRESS => "DB17200_MAINTENANCE_SEQUENCE".MAINTENANCE_IN_PROGRESS[58]);
END_REGION

REGION Network 64: ACTION IN MEDICOAT LINE 3 UNIT 2
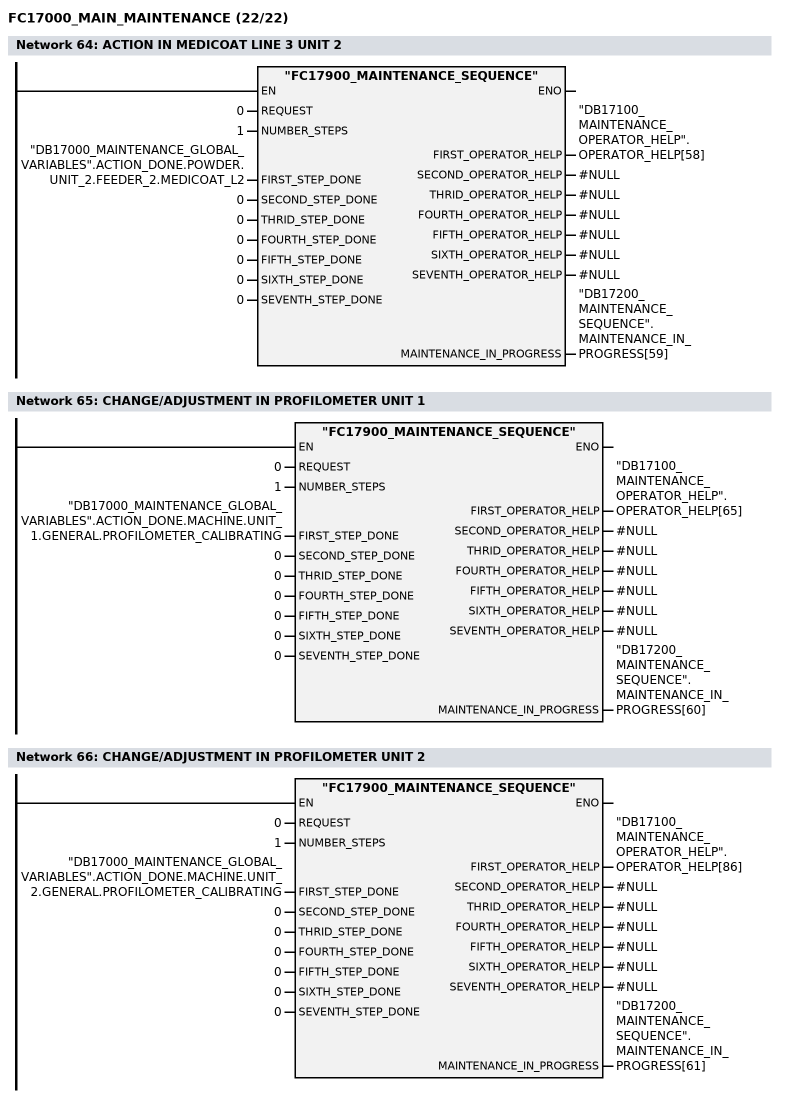
   RUNG wire#powerrail
      "FC17900_MAINTENANCE_SEQUENCE"(REQUEST := 0, NUMBER_STEPS := 1, FIRST_STEP_DONE := "DB17000_MAINTENANCE_GLOBAL_VARIABLES".ACTION_DONE.POWDER.UNIT_2.FEEDER_2.MEDICOAT_L2, SECOND_STEP_DONE := 0, THRID_STEP_DONE := 0, FOURTH_STEP_DONE := 0, FIFTH_STEP_DONE := 0, SIXTH_STEP_DONE := 0, SEVENTH_STEP_DONE := 0, FIRST_OPERATOR_HELP => "DB17100_MAINTENANCE_OPERATOR_HELP".OPERATOR_HELP[58], SECOND_OPERATOR_HELP => #NULL, THRID_OPERATOR_HELP => #NULL, FOURTH_OPERATOR_HELP => #NULL, FIFTH_OPERATOR_HELP => #NULL, SIXTH_OPERATOR_HELP => #NULL, SEVENTH_OPERATOR_HELP => #NULL, MAINTENANCE_IN_PROGRESS => "DB17200_MAINTENANCE_SEQUENCE".MAINTENANCE_IN_PROGRESS[59])
   END_RUNG
   // the same network as SCL:
   "FC17900_MAINTENANCE_SEQUENCE"(REQUEST := 0,
                           NUMBER_STEPS := 1,
                           FIRST_STEP_DONE := "DB17000_MAINTENANCE_GLOBAL_VARIABLES".ACTION_DONE.POWDER.UNIT_2.FEEDER_2.MEDICOAT_L2,
                           SECOND_STEP_DONE := 0,
                           THRID_STEP_DONE := 0,
                           FOURTH_STEP_DONE := 0,
                           FIFTH_STEP_DONE := 0,
                           SIXTH_STEP_DONE := 0,
                           SEVENTH_STEP_DONE := 0,
                           FIRST_OPERATOR_HELP => "DB17100_MAINTENANCE_OPERATOR_HELP".OPERATOR_HELP[58],
                           SECOND_OPERATOR_HELP => #NULL,
                           THRID_OPERATOR_HELP => #NULL,
                           FOURTH_OPERATOR_HELP => #NULL,
                           FIFTH_OPERATOR_HELP => #NULL,
                           SIXTH_OPERATOR_HELP => #NULL,
                           SEVENTH_OPERATOR_HELP => #NULL,
                           MAINTENANCE_IN_PROGRESS => "DB17200_MAINTENANCE_SEQUENCE".MAINTENANCE_IN_PROGRESS[59]);
END_REGION

REGION Network 65: CHANGE/ADJUSTMENT IN PROFILOMETER UNIT 1
   RUNG wire#powerrail
      "FC17900_MAINTENANCE_SEQUENCE"(REQUEST := 0, NUMBER_STEPS := 1, FIRST_STEP_DONE := "DB17000_MAINTENANCE_GLOBAL_VARIABLES".ACTION_DONE.MACHINE.UNIT_1.GENERAL.PROFILOMETER_CALIBRATING, SECOND_STEP_DONE := 0, THRID_STEP_DONE := 0, FOURTH_STEP_DONE := 0, FIFTH_STEP_DONE := 0, SIXTH_STEP_DONE := 0, SEVENTH_STEP_DONE := 0, FIRST_OPERATOR_HELP => "DB17100_MAINTENANCE_OPERATOR_HELP".OPERATOR_HELP[65], SECOND_OPERATOR_HELP => #NULL, THRID_OPERATOR_HELP => #NULL, FOURTH_OPERATOR_HELP => #NULL, FIFTH_OPERATOR_HELP => #NULL, SIXTH_OPERATOR_HELP => #NULL, SEVENTH_OPERATOR_HELP => #NULL, MAINTENANCE_IN_PROGRESS => "DB17200_MAINTENANCE_SEQUENCE".MAINTENANCE_IN_PROGRESS[60])
   END_RUNG
   // the same network as SCL:
   "FC17900_MAINTENANCE_SEQUENCE"(REQUEST := 0,
                           NUMBER_STEPS := 1,
                           FIRST_STEP_DONE := "DB17000_MAINTENANCE_GLOBAL_VARIABLES".ACTION_DONE.MACHINE.UNIT_1.GENERAL.PROFILOMETER_CALIBRATING,
                           SECOND_STEP_DONE := 0,
                           THRID_STEP_DONE := 0,
                           FOURTH_STEP_DONE := 0,
                           FIFTH_STEP_DONE := 0,
                           SIXTH_STEP_DONE := 0,
                           SEVENTH_STEP_DONE := 0,
                           FIRST_OPERATOR_HELP => "DB17100_MAINTENANCE_OPERATOR_HELP".OPERATOR_HELP[65],
                           SECOND_OPERATOR_HELP => #NULL,
                           THRID_OPERATOR_HELP => #NULL,
                           FOURTH_OPERATOR_HELP => #NULL,
                           FIFTH_OPERATOR_HELP => #NULL,
                           SIXTH_OPERATOR_HELP => #NULL,
                           SEVENTH_OPERATOR_HELP => #NULL,
                           MAINTENANCE_IN_PROGRESS => "DB17200_MAINTENANCE_SEQUENCE".MAINTENANCE_IN_PROGRESS[60]);
END_REGION

REGION Network 66: CHANGE/ADJUSTMENT IN PROFILOMETER UNIT 2
   RUNG wire#powerrail
      "FC17900_MAINTENANCE_SEQUENCE"(REQUEST := 0, NUMBER_STEPS := 1, FIRST_STEP_DONE := "DB17000_MAINTENANCE_GLOBAL_VARIABLES".ACTION_DONE.MACHINE.UNIT_2.GENERAL.PROFILOMETER_CALIBRATING, SECOND_STEP_DONE := 0, THRID_STEP_DONE := 0, FOURTH_STEP_DONE := 0, FIFTH_STEP_DONE := 0, SIXTH_STEP_DONE := 0, SEVENTH_STEP_DONE := 0, FIRST_OPERATOR_HELP => "DB17100_MAINTENANCE_OPERATOR_HELP".OPERATOR_HELP[86], SECOND_OPERATOR_HELP => #NULL, THRID_OPERATOR_HELP => #NULL, FOURTH_OPERATOR_HELP => #NULL, FIFTH_OPERATOR_HELP => #NULL, SIXTH_OPERATOR_HELP => #NULL, SEVENTH_OPERATOR_HELP => #NULL, MAINTENANCE_IN_PROGRESS => "DB17200_MAINTENANCE_SEQUENCE".MAINTENANCE_IN_PROGRESS[61])
   END_RUNG
   // the same network as SCL:
   "FC17900_MAINTENANCE_SEQUENCE"(REQUEST := 0,
                           NUMBER_STEPS := 1,
                           FIRST_STEP_DONE := "DB17000_MAINTENANCE_GLOBAL_VARIABLES".ACTION_DONE.MACHINE.UNIT_2.GENERAL.PROFILOMETER_CALIBRATING,
                           SECOND_STEP_DONE := 0,
                           THRID_STEP_DONE := 0,
                           FOURTH_STEP_DONE := 0,
                           FIFTH_STEP_DONE := 0,
                           SIXTH_STEP_DONE := 0,
                           SEVENTH_STEP_DONE := 0,
                           FIRST_OPERATOR_HELP => "DB17100_MAINTENANCE_OPERATOR_HELP".OPERATOR_HELP[86],
                           SECOND_OPERATOR_HELP => #NULL,
                           THRID_OPERATOR_HELP => #NULL,
                           FOURTH_OPERATOR_HELP => #NULL,
                           FIFTH_OPERATOR_HELP => #NULL,
                           SIXTH_OPERATOR_HELP => #NULL,
                           SEVENTH_OPERATOR_HELP => #NULL,
                           MAINTENANCE_IN_PROGRESS => "DB17200_MAINTENANCE_SEQUENCE".MAINTENANCE_IN_PROGRESS[61]);
END_REGION
END_FUNCTION
